(* Logix 5000 project; controller corte_tubos Emulate 5570 rev 32.11; software revision 32.00 *)

TASK MainTask (continuous, watchdog 500 ms) : MainProgram

MODULES
   Local : Emulate 5570 (ICP 2, rev 32.11)
      I_O : vendor 1 type 0 code 15 (ICP 3, rev 1.1, Output RPI 50 ms)
END_MODULES

PROGRAM MainProgram   (* main routine MainRoutine *)
VAR
   Action_000 : SFC_ACTION := (Status := 16#c020_0000, A := 1, Q := 1, PauseTimer := 1, Count := 1);
   Action_001 : SFC_ACTION := (Status := 16#0020_0000, PauseTimer := 1);
   Action_002 : SFC_ACTION := (Status := 16#0020_0000, PauseTimer := 1);
   Action_003 : SFC_ACTION := (Status := 16#0020_0000, PauseTimer := 1);
   Action_004 : SFC_ACTION := (Status := 16#0020_0000, PauseTimer := 1);
   Action_005 : SFC_ACTION := (Status := 16#0020_0000, PauseTimer := 1);
   Action_006 : SFC_ACTION := (Status := 16#0020_0000, PauseTimer := 1);
   Action_007 : SFC_ACTION := (Status := 16#0020_0000, PauseTimer := 1);
   Action_008 : SFC_ACTION := (Status := 16#0020_0000, PauseTimer := 1);
   Action_009 : SFC_ACTION := (Status := 16#0020_0000, PauseTimer := 1);
   Action_010 : SFC_ACTION := (Status := 16#0020_0000, PauseTimer := 1);
   Action_011 : SFC_ACTION := (Status := 16#0020_0000, PauseTimer := 1);
   Action_012 : SFC_ACTION := (Status := 16#0020_0000, PauseTimer := 1);
   Action_013 : SFC_ACTION := (Status := 16#0020_0000, PauseTimer := 1);
   Action_014 : SFC_ACTION := (Status := 16#0020_0000, PauseTimer := 1);
   Action_015 : SFC_ACTION := (Status := 16#0020_0000, PauseTimer := 1);
   Action_016 : SFC_ACTION := (Status := 16#0020_0000, PauseTimer := 1);
   Action_017 : SFC_ACTION := (Status := 16#0020_0000, PauseTimer := 1);
   Action_018 : SFC_ACTION := (Status := 16#0020_0000, PauseTimer := 1);
   Action_019 : SFC_ACTION := (Status := 16#0020_0000, PauseTimer := 1);
   Action_020 : SFC_ACTION := (Status := 16#0020_0000, PauseTimer := 1);
   Action_021 : SFC_ACTION := (Status := 16#0020_0000, PauseTimer := 1);
   Action_022 : SFC_ACTION := (Status := 16#0020_0000, PauseTimer := 1);
   Action_023 : SFC_ACTION := (Status := 16#0020_0000, PauseTimer := 1);
   Action_029 : SFC_ACTION := (Status := 16#0020_0000, PauseTimer := 1);
   B : BOOL;
   COUNTER : DINT;   // Contador de piezas
   DET_TUB : BOOL;   // Detección de tubo
   H1 : BOOL;   // Indicador de selección de tubo. Arranque
   H2 : BOOL;   // Indicación de pieza en proceso
   H3 : BOOL;
   L1 : BOOL;
   L10 : BOOL;
   L11 : BOOL;
   L12 : BOOL;
   L2 : BOOL;
   L3 : BOOL;
   L4 : BOOL;
   L5 : BOOL;
   L6 : BOOL;
   L7 : BOOL;
   L8 : BOOL;
   L9 : BOOL;
   LC : DINT;
   LR : DINT;   // Longitud de referencia
   Motor : BOOL;   // Control de encendido del motor de corte
   n : DINT := 6000;
   RESET : BOOL;
   S1 : BOOL;
   S2 : BOOL := 1;
   S3 : BOOL;
   S4 : BOOL := 1;
   S5 : BOOL;
   S6 : BOOL;
   S7 : BOOL := 1;
   Start : BOOL;
   Step_000 : SFC_STEP := (Status := 16#a820_0201, X := 1, SA := 1, DN := 1, PauseTimer := 1, T := 371150, TMax := 371150, Count := 1);
   Step_001 : SFC_STEP := (Status := 16#0020_0001, PauseTimer := 1);
   Step_002 : SFC_STEP := (Status := 16#0020_0001, PauseTimer := 1);
   Step_003 : SFC_STEP := (Status := 16#0020_0001, PauseTimer := 1, PRE := 200);
   Step_004 : SFC_STEP := (Status := 16#0020_0001, PauseTimer := 1);
   Step_005 : SFC_STEP := (Status := 16#0020_0000, PauseTimer := 1);
   Step_006 : SFC_STEP := (Status := 16#0020_0001, PauseTimer := 1);
   Step_007 : SFC_STEP := (Status := 16#0020_0001, PauseTimer := 1, PRE := 500);
   Step_008 : SFC_STEP := (Status := 16#0020_0001, PauseTimer := 1);
   Step_009 : SFC_STEP := (Status := 16#0020_0001, PauseTimer := 1);
   Step_010 : SFC_STEP := (Status := 16#0020_0001, PauseTimer := 1);
   Step_011 : SFC_STEP := (Status := 16#0020_0001, PauseTimer := 1);
   Step_012 : SFC_STEP := (Status := 16#0020_0001, PauseTimer := 1, PRE := 1000);
   Step_013 : SFC_STEP := (Status := 16#0020_0001, PauseTimer := 1, PRE := 1000);
   Step_014 : SFC_STEP := (Status := 16#0020_0001, PauseTimer := 1);
   Step_015 : SFC_STEP := (Status := 16#0020_0001, PauseTimer := 1);
   Step_016 : SFC_STEP := (Status := 16#0020_0001, PauseTimer := 1);
   Step_017 : SFC_STEP := (Status := 16#0020_0000, PauseTimer := 1);
   Stop : BOOL;
   Stop_Alarm : BOOL;
   Tran_000 : BOOL;
   Tran_001 : BOOL;
   Tran_002 : BOOL;
   Tran_003 : BOOL;
   Tran_004 : BOOL;
   Tran_005 : BOOL;
   Tran_006 : BOOL;
   Tran_007 : BOOL;
   Tran_008 : BOOL;
   Tran_009 : BOOL;
   Tran_010 : BOOL;
   Tran_011 : BOOL;
   Tran_012 : BOOL;
   Tran_013 : BOOL;
   Tran_014 : BOOL;
   Tran_015 : BOOL;
   Tran_016 : BOOL;
   Tran_017 : BOOL;
   Tran_018 : BOOL;
   Tran_019 : BOOL;
   Tran_020 : BOOL;
   Tran_021 : BOOL;
   Tran_022 : BOOL;
   Tran_023 : BOOL;
   Tran_024 : BOOL;
   Tran_025 : BOOL;
   Tran_026 : BOOL;
   Tran_027 : BOOL;
   Tran_028 : BOOL;
   Tran_029 : BOOL;
   Tran_030 : BOOL;
   Tran_031 : BOOL;
   Tran_032 : BOOL;
   Tran_033 : BOOL;
   Tran_034 : BOOL;
   Tran_035 : BOOL;
   Tran_036 : BOOL;
   Tran_037 : BOOL;
   Tran_038 : BOOL;
   Tran_039 : BOOL;
   Tran_040 : BOOL;
   Tran_041 : BOOL;
   Tran_042 : BOOL;
   Tran_043 : BOOL;
   Tran_044 : BOOL;
   Tran_045 : BOOL;
   Tran_046 : BOOL;
   Tran_047 : BOOL;
   Tran_048 : BOOL;
   Y1 : BOOL := 1;
   Y2 : BOOL;
   Y3 : BOOL := 1;
   Y4 : BOOL;
   Y5 : BOOL := 1;
   Y6 : BOOL;
END_VAR

ROUTINE calcular_parametros   (* structured text *)
   if L1 then
   	LC := 115;
   elsif L2 then
   	LC := 540;
   elsif L3 then
   	LC := 600;
   elsif L4 then
   	LC := 69;
   elsif L5 then
   	LC := 200;
   elsif L6 then
   	LC := 430;
   elsif L7 then
   	LC := 430;
   elsif L8 then
   	LC := 450;
   elsif L9 then
   	LC := 950;
   elsif L10 then
   	LC := 950;
   elsif L11 then
   	LC := 400;
   elsif L12 then
   	LC := 400;
   end_if;
   
   if LC <> 0 then
   	B := 1;
   	n:=6000/LC;
   end_if;
END_ROUTINE

ROUTINE config_inicial   (* structured text *)
   Y1:=0;
   Y2[:=]1;
   Y3:=0;
   Y4[:=]1;
   Y5[:=]1;
   Y6:=0;
   LC := 0;
   n := 0;
   H1 := 0;
   Motor := 0;
   COUNTER := 0;
   DET_TUB := 0;
   LR := 0;
   H2 := 0;
   H3 := 0;
   B := 0;
END_ROUTINE

ROUTINE Grafcet_general   (* sequential function chart *)
// secuencia de corte general
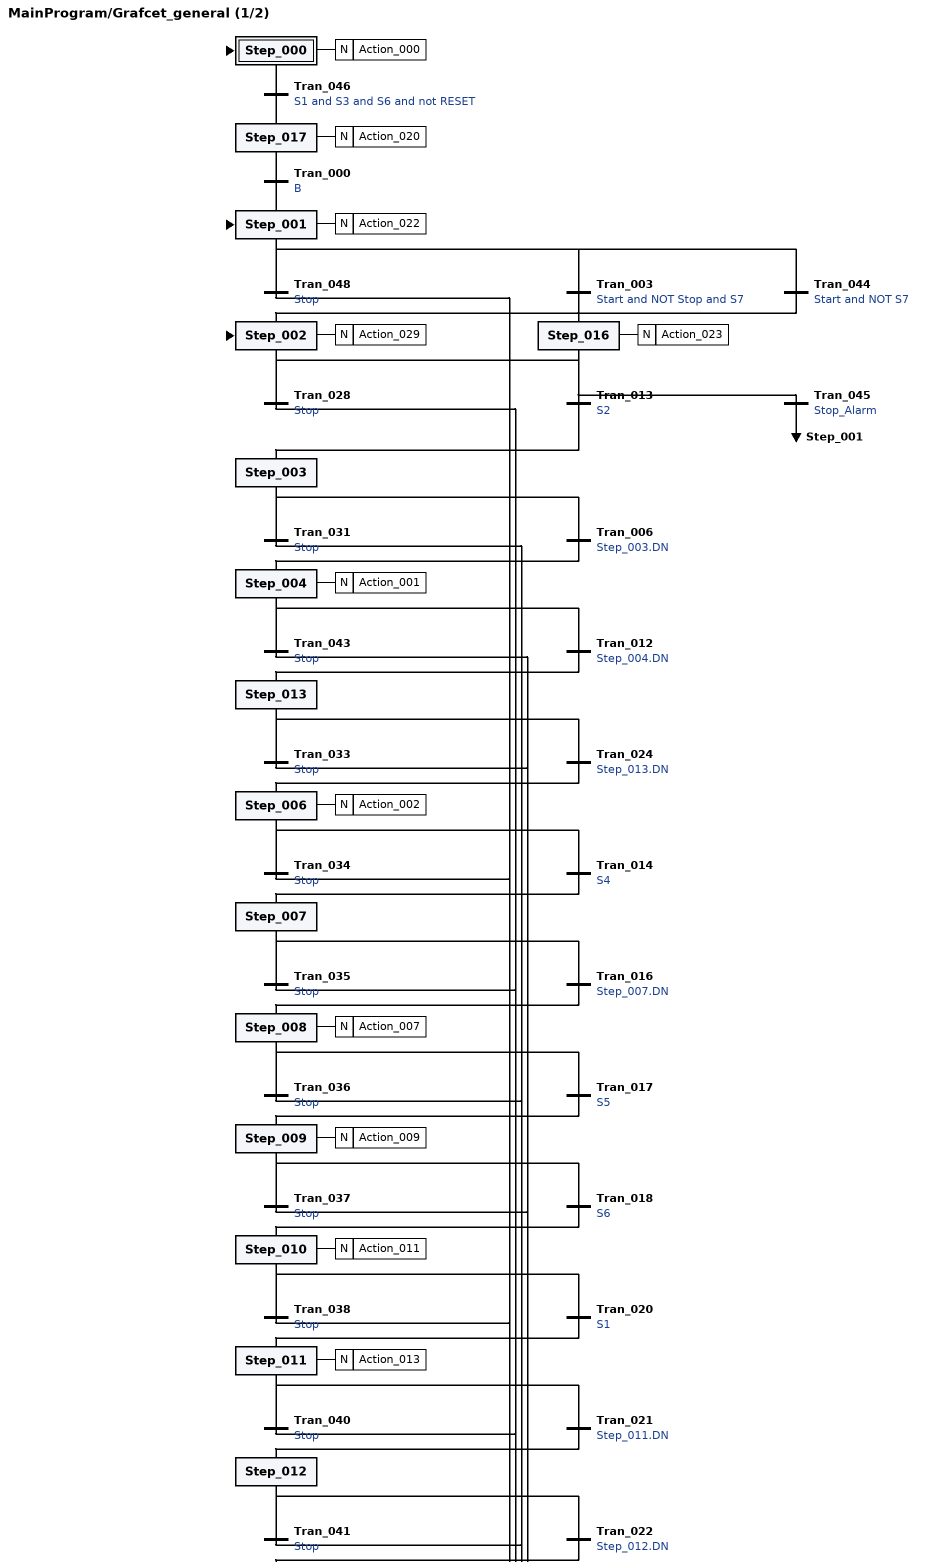
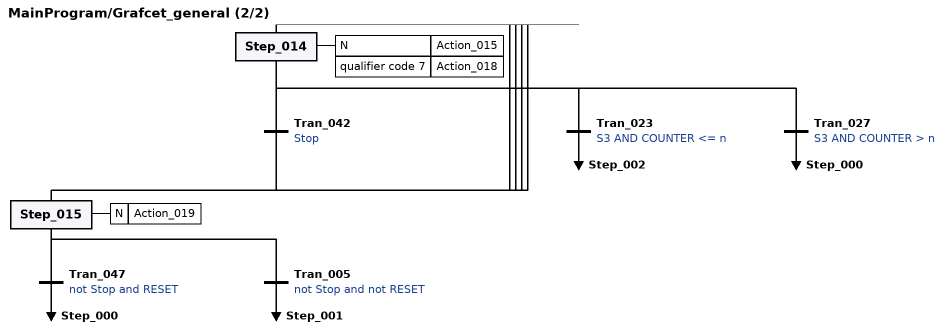
   INITIAL_STEP Step_000:
      ACTION Action_000 (N):
         JSR(config_inicial);
      END_ACTION
   END_STEP
   TRANSITION Tran_046 FROM Step_000 TO Step_017
      := S1 and S3 and S6 and not RESET
   END_TRANSITION
   STEP Step_015:
      ACTION Action_019 (N):
         H3 := 1;
         H2 := 0;
         H1 := 0;
         Y2 [:=] 1;
         Y4 [:=] 1;
         Y5 [:=] 1;
      END_ACTION
   END_STEP
   STEP Step_017:
      ACTION Action_020 (N):
         JSR(calcular_parametros);
      END_ACTION
   END_STEP
   TRANSITION Tran_047 FROM Step_015 TO Step_000
      := not Stop and RESET
         
   END_TRANSITION
   TRANSITION Tran_005 FROM Step_015 TO Step_001
      := not Stop and not RESET
   END_TRANSITION
   TRANSITION Tran_000 FROM Step_017 TO Step_001
      := B
   END_TRANSITION
   STEP Step_001:
      ACTION Action_022 (N):
         H1 := 1;
         H3 := 0;
      END_ACTION
   END_STEP
   TRANSITION Tran_048 FROM Step_001 TO Step_015
      := Stop
   END_TRANSITION
   TRANSITION Tran_003 FROM Step_001 TO Step_002
      := Start and NOT Stop and S7
   END_TRANSITION
   TRANSITION Tran_044 FROM Step_001 TO Step_016
      := Start and NOT S7
   END_TRANSITION
   STEP Step_016:
      ACTION Action_023 (N):
         H3 := 1;
         H2 := 0;
         H1 := 0;
      END_ACTION
   END_STEP
   STEP Step_002:
      ACTION Action_029 (N):
         Y1 [:=] 1;
         Motor := 1;
         H1 := 0;
         H2 := 1;
      END_ACTION
   END_STEP
   TRANSITION Tran_045 FROM Step_016 TO Step_001
      := Stop_Alarm
   END_TRANSITION
   TRANSITION Tran_028 FROM Step_002 TO Step_015
      := Stop
   END_TRANSITION
   TRANSITION Tran_013 FROM Step_002 TO Step_003
      := S2
   END_TRANSITION
   STEP Step_003:
   END_STEP
   TRANSITION Tran_031 FROM Step_003 TO Step_015
      := Stop
   END_TRANSITION
   TRANSITION Tran_006 FROM Step_003 TO Step_004
      := Step_003.DN
   END_TRANSITION
   STEP Step_004:
      ACTION Action_001 (N):
         LR := LC;
      END_ACTION
   END_STEP
   TRANSITION Tran_043 FROM Step_004 TO Step_015
      := Stop
   END_TRANSITION
   TRANSITION Tran_012 FROM Step_004 TO Step_013
      := Step_004.DN
   END_TRANSITION
   STEP Step_013:
   END_STEP
   TRANSITION Tran_033 FROM Step_013 TO Step_015
      := Stop
   END_TRANSITION
   TRANSITION Tran_024 FROM Step_013 TO Step_006
      := Step_013.DN
   END_TRANSITION
   STEP Step_006:
      ACTION Action_002 (N):
         Y3 [:=] 1;
         
      END_ACTION
   END_STEP
   TRANSITION Tran_034 FROM Step_006 TO Step_015
      := Stop
   END_TRANSITION
   TRANSITION Tran_014 FROM Step_006 TO Step_007
      := S4
   END_TRANSITION
   STEP Step_007:
   END_STEP
   TRANSITION Tran_035 FROM Step_007 TO Step_015
      := Stop
   END_TRANSITION
   TRANSITION Tran_016 FROM Step_007 TO Step_008
      := Step_007.DN
   END_TRANSITION
   STEP Step_008:
      ACTION Action_007 (N):
         Y6 [:=] 1;
      END_ACTION
   END_STEP
   TRANSITION Tran_036 FROM Step_008 TO Step_015
      := Stop
   END_TRANSITION
   TRANSITION Tran_017 FROM Step_008 TO Step_009
      := S5
   END_TRANSITION
   STEP Step_009:
      ACTION Action_009 (N):
         Y5 [:=] 1;
      END_ACTION
   END_STEP
   TRANSITION Tran_037 FROM Step_009 TO Step_015
      := Stop
   END_TRANSITION
   TRANSITION Tran_018 FROM Step_009 TO Step_010
      := S6
   END_TRANSITION
   STEP Step_010:
      ACTION Action_011 (N):
         Y2 [:=] 1;
      END_ACTION
   END_STEP
   TRANSITION Tran_038 FROM Step_010 TO Step_015
      := Stop
   END_TRANSITION
   TRANSITION Tran_020 FROM Step_010 TO Step_011
      := S1
   END_TRANSITION
   STEP Step_011:
      ACTION Action_013 (N):
         LR := 0;
         
      END_ACTION
   END_STEP
   TRANSITION Tran_040 FROM Step_011 TO Step_015
      := Stop
   END_TRANSITION
   TRANSITION Tran_021 FROM Step_011 TO Step_012
      := Step_011.DN
   END_TRANSITION
   STEP Step_012:
   END_STEP
   TRANSITION Tran_041 FROM Step_012 TO Step_015
      := Stop
   END_TRANSITION
   TRANSITION Tran_022 FROM Step_012 TO Step_014
      := Step_012.DN
   END_TRANSITION
   STEP Step_014:
      ACTION Action_015 (N):
         Y4 [:=] 1;
         DET_TUB [:=] 1;
      END_ACTION
      ACTION Action_018 (qualifier code 7):
         COUNTER := COUNTER + 1;
      END_ACTION
   END_STEP
   TRANSITION Tran_042 FROM Step_014 TO Step_015
      := Stop
   END_TRANSITION
   TRANSITION Tran_023 FROM Step_014 TO Step_002
      := S3 AND COUNTER <= n
   END_TRANSITION
   TRANSITION Tran_027 FROM Step_014 TO Step_000
      := S3 AND COUNTER > n
   END_TRANSITION
END_ROUTINE

ROUTINE MainRoutine   (* ladder *)
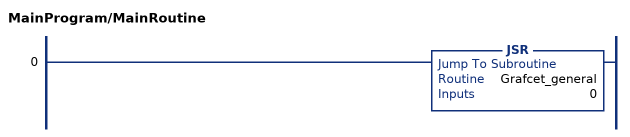
   0: JSR(Grafcet_general,0);
END_ROUTINE
END_PROGRAM
